# EPICS substitutions: src/main/epics/tspd-adqApp/Db/tspd-adq.substitutions
file ADQDevice.template
{
    pattern { INFO,  INFO_NELM }
            { INFO,  32        }
}

file ADQAIChannelGroup.template
{
    pattern { GRP }
            { COM }
}

file ADQAIChannel.template
{
    pattern { GRP,  CH  }
            { COM,  CH0 }
            { COM,  CH1 }
            { COM,  CH2 }
            { COM,  CH3 }
}
